(* CoDeSys 2.3 export: ETAGE_3.EXP *)

(* POU Initialisation_Standby/ETAGE_3, SFC *)
PROGRAM ETAGE_3
VAR
END_VAR
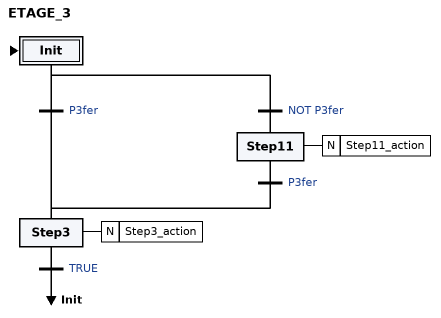
INITIAL_STEP Init:
END_STEP
TRANSITION FROM Init TO Step3 := P3fer;
END_TRANSITION
TRANSITION FROM Init TO Step11 := NOT P3fer;
END_TRANSITION
STEP Step11:
	Step11_action(N);
END_STEP
TRANSITION FROM Step11 TO Step3 := P3fer;
END_TRANSITION
STEP Step3:
	Step3_action(N);
END_STEP
TRANSITION FROM Step3 TO Init := TRUE;
END_TRANSITION

ACTION Step11_action:
F3:=TRUE;
END_ACTION

ACTION Step3_action:
F3:=FALSE;
END_ACTION
END_PROGRAM
